PROGRAM MAIN
VAR
END_VAR

TestProgram();

END_PROGRAM

(* stored: Version 1.1.0.1, ProductVersion 3.1.4022.10
   POU MAIN: Id {b151b296-7c6d-406f-b4d2-3b600f7011ad}, SpecialFunc None *)
